{attribute 'GeneratedUsingTerminal: EL3011-0000-0018'}
{attribute addProperty BoxType "EL3011-0000-0018"}
{attribute addProperty Id "AI_StandardAT %I*AI_Standard_4A3944819WcStateAT %I*WcState_9091E0EB2InfoDataAT %I*InfoData_23CBA8372"}
{attribute addProperty CRC "3100264523"}
{attribute addProperty Size "13"}
TYPE EL3011_B8CA484B EXTENDS TcoIo.EtcSlaveTerminalBase_947E5A46 :
STRUCT
	{attribute addProperty Name "AI_Standard"}
	AI_Standard : AI_Standard_4A394481;
	{attribute addProperty Name "WcState"}
	WcState : TcoIo.WcState_9091E0EB;
	{attribute addProperty Name "InfoData"}
	InfoData : InfoData_23CBA837;
END_STRUCT
END_TYPE

(* stored: Version 1.2.0.0, ProductVersion 3.1.4024.9
   DUT EL3011_B8CA484B: Id {5da3ccaa-19c2-0293-3d0b-71dec7551672} *)
